(* IEC 61131-3 sources: Industry-PLC-LLM/data/PLCBEAD_repo/PLCBEAD_PLCEmbed-main/PLC-BEAD/Source/GEB/Network_TN_SC_SHADOW_ATTR, 1 file *)

(* ---- TN_SC_SHADOW_ATTR.ST ---- *)
FUNCTION TN_SC_SHADOW_ATTR:BYTE

	VAR_INPUT
		Iby_ATTR :	BYTE;
	END_VAR

	TN_SC_SHADOW_ATTR := ((Iby_ATTR AND BYTE#2#11110000) OR BYTE#2#00001000);

END_FUNCTION

PROGRAM program0
	VAR
		Iby_ATTR :	BYTE;
		CEIL5_OUT : BYTE;
	END_VAR

  	CEIL5_OUT := TN_SC_SHADOW_ATTR(Iby_ATTR);
END_PROGRAM
